{attribute 'TcGenerated'}
{attribute 'no-analysis'}
{attribute 'linkalways'}
// This function has been automatically generated from the project information.
VAR_GLOBAL CONSTANT
	{attribute 'const_non_replaced'}
	stLibVersion_TestHarnessCore : ST_LibVersion := (iMajor := 0, iMinor := 0, iBuild := 4, iRevision := 0, nFlags := 0, sVersion := '0.0.4');
END_VAR

(* stored: Version 1.1.0.1, ProductVersion 3.1.4026.18
   GVL Global_Version: Id {2cffabf8-03a0-4a99-9503-257d0a2e6977} *)
